Omron CX-Programmer project NewProject (CX-Programmer 9.75)

# PLC NewPLC1: CP1H XA

## Global symbols (name address type ; comment)
0.00 BOOL  ; Input
0.01 BOOL  ; Reset
0.02 BOOL  ; S_5cm
0.03 BOOL  ; S_15cm
0.04 BOOL  ; S_25cm
0.05 BOOL  ; Sesnor CNT
100.00 BOOL  ; Lampu 1
100.01 BOOL  ; Conveyor
100.02 BOOL  ; Indikator 5cm
100.03 BOOL  ; Indikator 15cm
100.04 BOOL  ; Indikator 25cm
100.05 BOOL  ; sirine
100.06 BOOL  ; conveyor2
100.07 BOOL  ; conveyor3
100.08 BOOL  ; conveyor4
100.09 BOOL  ; Sirine 2
200.00 BOOL  ; pneumatik 5 cm
200.01 BOOL  ; pneumatic
200.02 BOOL  ; stopper
200.03 BOOL  ; pneumatik 15 cm
200.04 BOOL  ; stopper
200.05 BOOL  ; pneumatik 25 cm
W0.00 BOOL  ; start
W0.01 BOOL  ; reset

## Program NewProgram1 (cyclic task 0)

### Section Section1

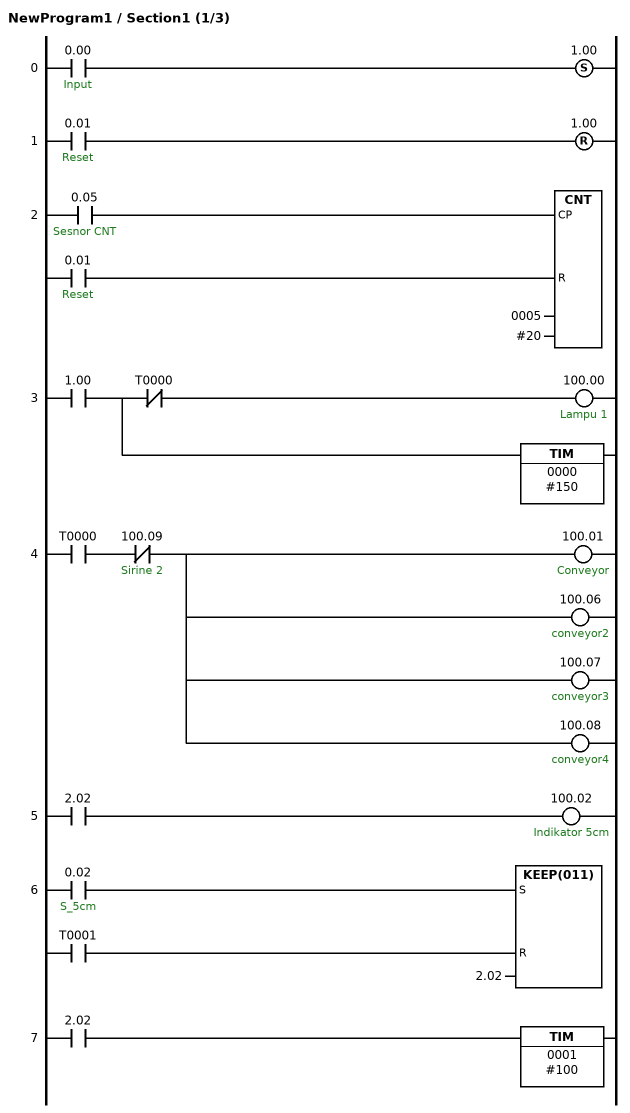
; rung 0
LD 0.00  ; Input
SET 1.00
; rung 1
LD 0.01  ; Reset
RSET 1.00
; rung 2
LD 0.05  ; Sesnor CNT
LD 0.01  ; Reset
CNT 0005 #20
; rung 3
LD 1.00
OUT TR0
ANDNOT T0000
OUT 100.00  ; Lampu 1
LD TR0
TIM 0000 #150
; rung 4
LD T0000
ANDNOT 100.09  ; Sirine 2
OUT 100.01  ; Conveyor
OUT 100.06  ; conveyor2
OUT 100.07  ; conveyor3
OUT 100.08  ; conveyor4
; rung 5
LD 2.02
OUT 100.02  ; Indikator 5cm
; rung 6
LD 0.02  ; S_5cm
LD T0001
KEEP(011) 2.02
; rung 7
LD 2.02
TIM 0001 #100

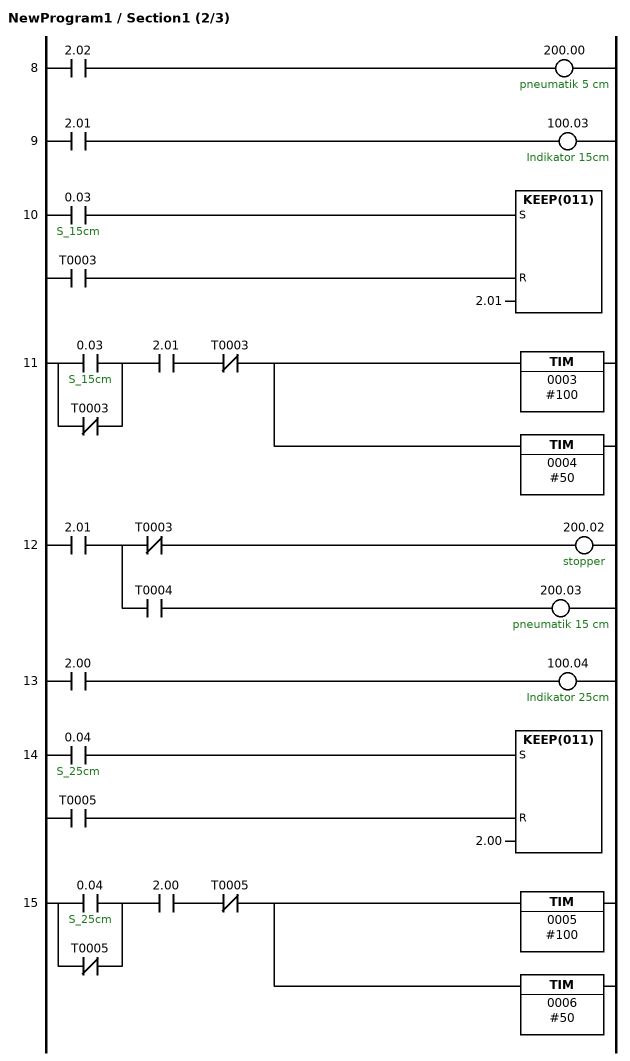
; rung 8
LD 2.02
OUT 200.00  ; pneumatik 5 cm
; rung 9
LD 2.01
OUT 100.03  ; Indikator 15cm
; rung 10
LD 0.03  ; S_15cm
LD T0003
KEEP(011) 2.01
; rung 11
LD 0.03  ; S_15cm
ORNOT T0003
AND 2.01
ANDNOT T0003
TIM 0003 #100
TIM 0004 #50
; rung 12
LD 2.01
OUT TR0
ANDNOT T0003
OUT 200.02  ; stopper
LD TR0
AND T0004
OUT 200.03  ; pneumatik 15 cm
; rung 13
LD 2.00
OUT 100.04  ; Indikator 25cm
; rung 14
LD 0.04  ; S_25cm
LD T0005
KEEP(011) 2.00
; rung 15
LD 0.04  ; S_25cm
ORNOT T0005
AND 2.00
ANDNOT T0005
TIM 0005 #100
TIM 0006 #50

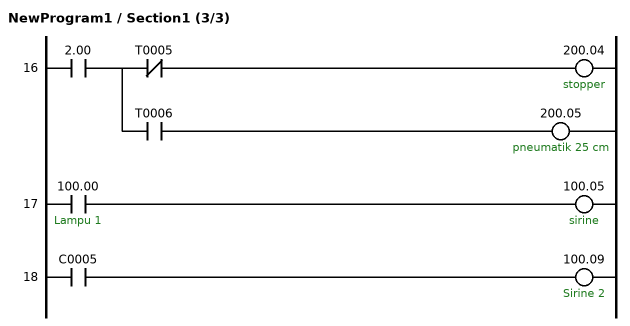
; rung 16
LD 2.00
OUT TR0
ANDNOT T0005
OUT 200.04  ; stopper
LD TR0
AND T0006
OUT 200.05  ; pneumatik 25 cm
; rung 17
LD 100.00  ; Lampu 1
OUT 100.05  ; sirine
; rung 18
LD C0005
OUT 100.09  ; Sirine 2

### Section END
; rung 0
END(001)